FUNCTION F_RotatePositionXY : HRESULT
VAR_INPUT
	fbPosition : REFERENCE TO Tc3_Physics.PositionXY;
	fRotate : LREAL; //[°]
END_VAR
VAR
	fRadius : LREAL;
	fPhi : LREAL;
	fNewPhi : LREAL;
END_VAR

IF NOT __ISVALIDREF(fbPosition) THEN
	F_RotatePositionXY := E_FAIL;
	RETURN;
END_IF

fRadius := fbPosition.GetRadius();
fPhi := fbPosition.GetPhi();

fNewPhi := MODABS((fPhi + fRotate), 360.0);

fbPosition.SetValuesRP(radius := fRadius, phi := fNewPhi);

END_FUNCTION

(* stored: Version 1.1.0.1, ProductVersion 3.1.4024.12
   POU F_RotatePositionXY: Id {d955eb06-90fc-423e-a240-9df928823a65}, SpecialFunc None *)
